// TIA Portal V20 export
TYPE "CMInterface_DI"
   STRUCT
      Input { ExternalAccessible := 'False'; ExternalVisible := 'False'; ExternalWritable := 'False'} : Bool;
   END_STRUCT;
END_TYPE
